PROGRAM PMPS_Arbiter
VAR
	
	getPosPtr	: POINTER TO T_HashTableEntry := 0;
	getBPStruct	:	ST_BeamParams;
	stOutputBP	:	ST_BeamParams; //Safest beam parameters from all in the assertion pool
	
	fbMachine	:	FB_MachineSimulator;
END_VAR



//Arbitrate
(*
This step cycles through every hash table entry, comparing
the beam parameters from each assertion to what we're planning
to assert.

The safer of the two parameters is kept so at the end we may
have a mix of beam parameters, the composition being safe for
all asserters.

*)

//Safest parameters to start
stOutputBP := F_SetBeamParams(
	fAtt := 100,
	fPP_mJ := 0,
	fLower_eV := 0,
	fUpper_eV := 1800
	);

fbBPAssertionPool.A_GetFirst( putPosPtr := 0, getPosPtr=>getPosPtr, getValue=>getBPStruct );
IF fbBPAssertionPool.bOk THEN
	
	//The first entry in the hash table is taken as the setting to arbitrate against
	stOutputBP := F_SetBeamParams(
		fAtt := getBPStruct.fAtt,
		fPP_mJ := getBPStruct.fPP_mJ,
		fLower_eV := getBPStruct.fLower_eV,
		fUpper_eV := getBPStruct.fUpper_eV
	);

	REPEAT
		fbBPAssertionPool.A_GetNext( putPosPtr := fbBPAssertionPool.getPosPtr , getPosPtr=>getPosPtr, getValue=>getBPStruct );
		IF fbBPAssertionPool.bOk THEN
			A_Arbitrate();
		END_IF
	UNTIL NOT fbBPAssertionPool.bOk
	END_REPEAT

END_IF

//Machine simulator
fbMachine(
	i_stAssertedParams := stOutputBP,
	q_stMachineParams => PMPS_GVL_BeamParams.stCurrentBeamParameters
	);

ACTION A_Arbitrate:

//Attenuation
//Add something here to register the key that won for each param
stOutputBP.fAtt := MAX(stOutputBP.fAtt, getBPStruct.fAtt);

//Pulse energy
stOutputBP.fPP_mJ := MIN(stOutputBP.fPP_mJ, getBPStruct.fPP_mJ);

stOutputBP.fLower_eV := MAX(stOutputBP.fLower_eV, getBPStruct.fLower_eV);
stOutputBP.fUpper_eV := MIN(stOutputBP.fUpper_eV, getBPStruct.fUpper_eV);
END_ACTION

END_PROGRAM

(* stored: Version 1.1.0.1, ProductVersion 3.1.4022.12
   POU PMPS_Arbiter: Id {91ae890b-11cc-4d41-83ec-edc5b802c784}, SpecialFunc None
   Action A_Arbitrate: Id {cd232571-a3df-0041-3bcc-1fe44a9b9a88} *)
